PROGRAM Test
VAR
END_VAR

END_PROGRAM

(* stored: Version 1.1.0.1, ProductVersion 3.1.4022.18
   POU Test: Id {05a7abdc-a21b-48aa-9907-14c130b4fdc8}, SpecialFunc None *)
